// TIA Portal project "TimerEContatori" (V20)

(* hardware
DEVICE "S7-1200 station_1"  S7-1200 Station
   slot 0: "Rack_0"  S7-1200 Rack  Rack  V1.0
   slot 1: "Playground_PLC"  CPU 1214C DC/DC/DC  6ES7 214-1AG40-0XB0  V4.7
   slot 3: "AQ 1x12BIT_1"  AQ1 signal board  6ES7 232-4HA30-0XB0  V1.0
*)

// ===== PLC "Playground_PLC"  CPU 1214C DC/DC/DC =====

VAR_GLOBAL   // PLC tag table "Default tag table"
   "BTN_BUZ" AT %M0.0 : Bool;
   "BTN_LAMP" AT %M0.1 : Bool;
   "BUZZ" AT %M0.2 : Bool;
   "LAMP" AT %M0.3 : Bool;
   "RESET_BUZ" AT %M0.4 : Bool;
   "RESET_LAMP" AT %M0.5 : Bool;
END_VAR

DATA_BLOCK "COUNTERS"   // DB4
{ S7_Optimized_Access := 'TRUE' }
VERSION : 0.1
   VAR
      BUZ_COUNTER : USInt := 6;
      LAMP_COUNTER : USInt := 7;
   END_VAR
BEGIN
END_DATA_BLOCK

DATA_BLOCK "TIMERS"   // DB5
{ S7_Optimized_Access := 'TRUE' }
VERSION : 0.1
   VAR
      BUZ_TIMER : Time := T#5S;
      LAMP_TIMER : Time := T#10S;
   END_VAR
BEGIN
END_DATA_BLOCK

// folder: System blocks/Program resources

DATA_BLOCK "IEC_Counter_0_DB_2"   // DB3
{ S7_Optimized_Access := 'TRUE' }
AUTHOR : Simatic
FAMILY : IEC
NAME : CNTR
VERSION : 1.0
// stored: InstanceOfName IEC_COUNTER
"IEC_COUNTER"
BEGIN
END_DATA_BLOCK

DATA_BLOCK "IEC_Timer_0_DB"   // DB6
{ S7_Optimized_Access := 'TRUE' }
AUTHOR : Simatic
FAMILY : IEC
NAME : IEC_TMR
VERSION : 1.0
// stored: InstanceOfName IEC_TIMER
"IEC_TIMER"
BEGIN
END_DATA_BLOCK

DATA_BLOCK "IEC_Counter_0_DB_3"   // DB7
{ S7_Optimized_Access := 'TRUE' }
AUTHOR : Simatic
FAMILY : IEC
NAME : CNTR
VERSION : 1.0
// stored: InstanceOfName IEC_COUNTER
"IEC_COUNTER"
BEGIN
END_DATA_BLOCK

DATA_BLOCK "IEC_Timer_0_DB_1"   // DB8
{ S7_Optimized_Access := 'TRUE' }
AUTHOR : Simatic
FAMILY : IEC
NAME : IEC_TMR
VERSION : 1.0
// stored: InstanceOfName IEC_TIMER
"IEC_TIMER"
BEGIN
END_DATA_BLOCK

// folder: (top level)

ORGANIZATION_BLOCK "Main"   // OB1, LAD, ProgramCycle
TITLE = "Main Program Sweep (Cycle)"
{ S7_Optimized_Access := 'TRUE' }
VERSION : 0.1
   VAR_INPUT
      Initial_Call : Bool;   // Initial call of this OB
      Remanence : Bool;   // =True, if remanent data are available
   END_VAR
BEGIN

REGION Network 1
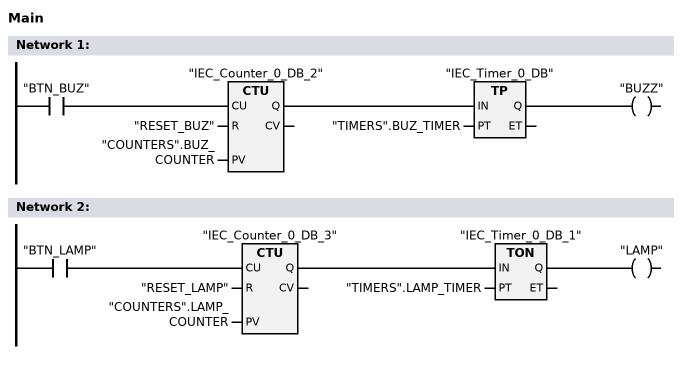
   "IEC_Counter_0_DB_2".CTU(CU := "BTN_BUZ", R := "RESET_BUZ", PV := "COUNTERS".BUZ_COUNTER);
   "IEC_Timer_0_DB".TP(IN := "IEC_Counter_0_DB_2".Q, PT := "TIMERS".BUZ_TIMER);
   "BUZZ" := "IEC_Timer_0_DB".Q;
END_REGION

REGION Network 2
   "IEC_Counter_0_DB_3".CTU(CU := "BTN_LAMP", R := "RESET_LAMP", PV := "COUNTERS".LAMP_COUNTER);
   "IEC_Timer_0_DB_1".TON(IN := "IEC_Counter_0_DB_3".Q, PT := "TIMERS".LAMP_TIMER);
   "LAMP" := "IEC_Timer_0_DB_1".Q;
END_REGION
END_ORGANIZATION_BLOCK